{attribute 'linkalways'} 
{attribute 'no_explicit_call' := 'This FB is a CLASS and must be accessed using methods or properties'}
{attribute 'enable_dynamic_creation'}
FUNCTION_BLOCK Node_ContainerType_Vector_Vector_TcVnPoint2_DINT EXTENDS Node
VAR
    out : _GUID;
END_VAR

METHOD PUBLIC  Clone : I_Node
VAR
	pNode : POINTER TO Node_ContainerType_Vector_Vector_TcVnPoint2_DINT;
END_VAR
pNode := __NEW(Node_ContainerType_Vector_Vector_TcVnPoint2_DINT);
Clone := pNode^;
END_METHOD

METHOD FB_init : BOOL
VAR_INPUT
	bInitRetains : BOOL; // if TRUE, the retain variables are initialized (warm start / cold start)
	bInCopyCode : BOOL;  // if TRUE, the instance afterwards gets moved into the copy code (online change)
END_VAR
AddOutput('out', out);
END_METHOD

METHOD PROTECTED OnExecute
out.Value := ContainerType_Vector_Vector_TcVnPoint2_DINT;
END_METHOD

END_FUNCTION_BLOCK

(* stored: Version 1.1.0.1, ProductVersion 3.1.4026.17
   POU Node_ContainerType_Vector_Vector_TcVnPoint2_DINT: Id {80ae5a47-7571-0d7d-0639-7d99df1d4d06}, SpecialFunc None
   Folder Constructor: Id {406a8818-3641-0a9c-0131-63c0efdf2400}
   Method Clone: Id {e2ecfe09-69d9-06a7-2737-38d453e82c06}
   Method FB_init: Id {714ad9cd-b59e-001a-25dc-36386224146b}
   Method OnExecute: Id {3b654a7b-51e4-0cc4-2fb6-ccc47135e503} *)
